TEXTLIST tlMissionIDs
  0 = 'NoMission_0'
  1 = 'ScrewMission_110'
  2 = 'StapleMission_120'
  3 = 'NailMission_130'
  4 = 'MillMissionCircle_140'
  5 = 'MillMissionRect_150'
  6 = 'MillMissionLine_160'
  7 = 'MillMissionCommonScrap_200'
  8 = 'MillMissionCommonNoScrap_210'
  9 = 'PickBoardMission_400'
  10 = 'PlaceBoardMissionAndScrew_401'
  11 = 'PlaceBoardMissionAndStaple_402'
  12 = 'PlaceBoardMissionAndNail_403'
  13 = 'GoToHomePosition_501'
  14 = 'GoToSafePosition_502'
  15 = 'LeaveTool_503'
  16 = 'GetBoardTool_504'
  17 = 'GetScrapTool_505'
  18 = 'GetScrewTool_506'
  19 = 'GetStapleTool_507'
  20 = 'GetNailTool_508'
   = ''
END_TEXTLIST

(* stored: Version 1.1.0.1, ProductVersion 3.1.4022.12
   TextList tlMissionIDs: Id {1c9c1b86-5c60-4941-8547-0e7eeb337c94} *)
